FUNCTION_BLOCK FB_MSF_Pistoni
VAR_INPUT
	bEnable	: BOOL;
	slot	: INT;
	iMotor	: INT;
END_VAR

VAR_IN_OUT
	
	st_In	:	ST_CSL_In;
	st_Params	: ST_CSL_Params;
	st_Out		: ST_CSL_Out;
	
END_VAR


VAR_OUTPUT
	
	
	
	eStep	: E_Step;		//current step of the state machine
	eErrStep : E_Step;  //step where an error was raised
	nErrid	: DINT;		//error identification code
	
	
	
	END_VAR
VAR
	bSensor: BOOL;
	bValve : BOOL;
	nStepSlot : INT;
	Timer_Pistons : TON();
	Error: DINT;
    

	bInitialized	: BOOL;		//FB initialization
	eNewStep : E_Step;			//request for a new step
	bEntryact	: 	BOOL;		//step entry action performed
		
END_VAR

(* initialization *)
IF NOT bInitialized THEN    
eNewstep := E_Step.NoStep;    
eStep := E_Step.Stop;    
bEntryact := FALSE;    
bInitialized := TRUE; 

ELSE   

(* forcing the error state *)	
(* disabled or faulty *)
IF NOT bEnable THEN
eNewstep := E_Step.NeOrError;

END_IF;

(* state change managementstate change management *)
IF eNewstep <> E_Step.NoStep THEN    
eStep := eNewstep;    
eNewstep := E_Step.NoStep;   
 bEntryact := FALSE;

END_IF;

// association of the motors and the sensors to the steps
CASE slot OF
	0:
		nStepSlot	:=	st_Params.StepNoSlot;	
	1:
		bValve:= st_Out.bValveSlot1;
		bSensor := st_In.bSlot1;
		nStepSlot := st_Params.StepSlot1;
	2:
		bValve:= st_Out.bValveSlot2;
		bSensor := st_In.bSlot2;
		nStepSlot := st_Params.StepSlot2;
	3:
		bValve:= st_Out.bValveSlot3;
		bSensor := st_In.bSlot3;
		nStepSlot := st_Params.StepSlot3;
END_CASE

(* input signal conditioning *)
Timer_Pistons (IN:= (iMotor = nStepSlot), PT := T#500MS);

// storing of the pieces
CASE eStep OF

// conveyor of the pieces
	E_Step.conveyor :
	
		(* body *)	
		st_Out.bMotor	:= TRUE;
		st_Out.bCompressor := TRUE;
		bValve 	:=	FALSE;	
		
		(* transition *)	
		IF bEnable THEN          
		 eNewstep := E_Step.NeOrError;        
		ELSE 
			IF  iMotor = nStepSlot THEN 
		eNewstep := E_Step.waiting;            
	
        END_IF;
	END_IF
	
	// waiting of the measure of the pieces color and number of steps
	E_Step.waiting :
	
		(* body *)
		st_Out.bMotor	:= FALSE;
		st_Out.bCompressor := TRUE;
		bValve 	:=	FALSE;	
		
		
		(* transition *)
		IF bEnable THEN          
		 eNewstep := E_Step.NeOrError;        
		ELSE 
			IF  Timer_Pistons.Q THEN 
		eNewstep := E_Step.piston;            
	
        END_IF;
	END_IF	
	
	// activation of the motors of the pistons.
	E_Step.piston :
		(* body *)
		st_Out.bMotor	:= FALSE;
		st_Out.bCompressor := TRUE;
		bValve 	:=	TRUE;	       
	
ELSE
	
// Error case
	eNewstep := E_Step.NeOrError;
	eErrStep := E_Step.Unknown;
	nErrId := -9; 	
		
		
END_CASE

 END_IF

END_FUNCTION_BLOCK

(* stored: Version 1.1.0.1, ProductVersion 3.1.4024.12
   POU FB_MSF_Pistoni: Id {78e36ba8-cb60-4537-88b2-3ff9943f6860}, SpecialFunc None *)
